# EPICS substitutions: db/ecmcEL9576.substitutions
file ecmcEcSlave.template
{
    pattern {}
            {}
}

file ecmcEL9576.template
{
	pattern {}
		    {}
}
